SUBAPPLICATION IE_UP (* Subapplication Type *)
  (* Standard: 61499-2 *)
  (* Version 1.0, 2023-02-06, franz *)
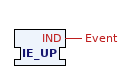
  EVENT_OUTPUT
    IND;
  END_EVENT
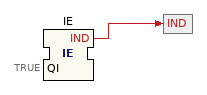
  FBS
    IE : IE(QI := TRUE);
  END_FBS
  EVENT_CONNECTIONS
    IE.IND TO IND;
  END_CONNECTIONS
END_SUBAPPLICATION
